(* Logix 5000 project; controller Line_Information_Standard vendor 1 type 14 code 151 rev 28.11; software revision 28.00 *)

TASK MainTask (continuous, watchdog 500 ms) : MainProgram

MODULES
   Local : vendor 1 type 14 code 151 (Compact 0, rev 28.11)
      Counters : Embedded (Compact 3, rev 1.1, Output RPI 20 ms)
      Analog_IO : Embedded (Compact 2, rev 1.1, Output RPI 80 ms)
      Discrete_IO : Embedded (Compact 1, rev 3.1, Output RPI 20 ms)
END_MODULES

TYPE ControlInterlock :   // Datatype for control interlocks to machines
STRUCT
   Connection : CONNECTION_STATUS;   // Machine connection status
   run : BOOL;   // OK to run machine
   jog : BOOL;   // OK to jog machine
   feed : BOOL;   // OK to feed machine
   commandRunSpeed : DINT;   // Commanded run speed
   commandJogSpeed : DINT;   // Commanded jog speed
   Time : DINT[7];   // Clock time
   MiscDINT : DINT[4];   // Miscellaneous digital values
   MiscREAL : REAL[4];   // Miscellaneous analog values
   MiscBOOL : BOOL[32];   // Miscellaneous bit values
END_STRUCT
END_TYPE

TYPE ConveyingControlInterlock :   // Datatype for control interlocks to conveying
STRUCT
   Connection : CONNECTION_STATUS;   // Machine connection status
   Running : BOOL[32];   // Machine running array
   Feeding : BOOL[32];   // Machine feeding array
   ProductIn : BOOL[32];   // Product in machine array
   CommandRunSpeed : DINT[64];   // Conveyor commanded run speed array
   Time : DINT[7];   // Clock time
   MiscDINT : DINT[8];   // Miscellaneous digital values
   MiscREAL : REAL[8];   // Miscellaneous analog values
   MiscBOOL : BOOL[64];   // Miscellaneous bit values
END_STRUCT
END_TYPE

TYPE ConveyingStatusInterlock :   // Datatype for status interlocks from conveying
STRUCT
   Connection : CONNECTION_STATUS;   // Machine connection status
   Faulted : BOOL[64];   // Conveyor faulted array
   Ready : BOOL[64];   // Conveyor ready array
   Running : BOOL[64];   // Conveyor running array
   Auto : BOOL[64];   // Conveyor in auto array
   Run : BOOL[32];   // OK to run machine array
   Feed : BOOL[32];   // OK to feed machine array
   ActualSpeed : DINT[64];   // Actual speed of conveyor array
   MiscDINT : DINT[8];   // Miscellaneous digital values
   MiscREAL : REAL[8];   // Miscellaneous analog values
   MiscBOOL : BOOL[64];   // Miscellaneous bit values
END_STRUCT
END_TYPE

TYPE LineInformation :   // Datatype for interfaces and displays
STRUCT
   Faults : BOOL[2048];   // Fault bit array
   MachineStatus : SINT[32];   // Machine statuses array
   MachineDown : BOOL[32];   // Machine down bit array
   BaseProductionCount : DINT[32];   // Base production counts array
   PackProductionCount : DINT[32];   // Package production counts array
   ActualBasePerPack : INT[32];   // Actual base per package multiplier array
   NominalBasePerPack : INT[32];   // Nominal base per package multiplier array
   ConveyorStatus : SINT[64];   // Conveyor statuses array
   Recipe : DINT[128];   // Recipe values
   Time : DINT[7];   // Clock time
   DST : SINT;   // Daylight saving time
   timeZone : SINT;   // Time zone UTC offset
   MiscDINT : DINT[8];   // Miscellaneous digital values
   MiscREAL : REAL[8];   // Miscellaneous analog values
   MiscBOOL : BOOL[64];   // Miscellaneous bit values
END_STRUCT
END_TYPE

TYPE MessageControlInterlock :   // Datatype for message control interlocks to machines
STRUCT
   Connection : SINT;   // Initial byte of memory to satisfy copy instruction
   run : BOOL;   // OK to run machine
   jog : BOOL;   // OK to jog machine
   feed : BOOL;   // OK to feed machine
   commandRunSpeed : DINT;   // Commanded run speed
   commandJogSpeed : DINT;   // Commanded jog speed
   Time : DINT[7];   // Clock time
   MiscDINT : DINT[4];   // Miscellaneous digital values
   MiscREAL : REAL[4];   // Miscellaneous analog values
   MiscBOOL : BOOL[32];   // Miscellaneous bit values
END_STRUCT
END_TYPE

TYPE MessageStatusInterlock :   // Datatype for message status interlocks from machines
STRUCT
   Connection : SINT;   // Initial byte of memory to satisfy copy instruction
   faulted : BOOL;   // Machine faulted
   ready : BOOL;   // Machine ready
   running : BOOL;   // Machine running
   jogging : BOOL;   // Machine jogging
   feeding : BOOL;   // Machine feeding
   productIn : BOOL;   // Product in machine
   actualSpeed : DINT;   // Actual speed of machine
   baseProductionCount : DINT;   // Base production count
   packProductionCount : DINT;   // Package production count
   basePerPack : INT;   // Base per package multiplier
   MiscDINT : DINT[4];   // Miscellaneous digital values
   MiscREAL : REAL[4];   // Miscellaneous analog values
   MiscBOOL : BOOL[32];   // Miscellaneous bit values
END_STRUCT
END_TYPE

TYPE StatusInterlock :   // Datatype for status interlocks from machines
STRUCT
   Connection : CONNECTION_STATUS;   // Machine connection status
   faulted : BOOL;   // Machine faulted
   ready : BOOL;   // Machine ready
   running : BOOL;   // Machine running
   jogging : BOOL;   // Machine jogging
   feeding : BOOL;   // Machine feeding
   productIn : BOOL;   // Product in machine
   actualSpeed : DINT;   // Actual speed of machine
   baseProductionCount : DINT;   // Base production count
   packProductionCount : DINT;   // Package production count
   basePerPack : INT;   // Base per package multiplier
   MiscDINT : DINT[4];   // Miscellaneous digital values
   MiscREAL : REAL[4];   // Miscellaneous analog values
   MiscBOOL : BOOL[32];   // Miscellaneous bit values
END_STRUCT
END_TYPE

VAR_GLOBAL   (* controller tags *)
   Clock : DINT[7] := ([0] := 2017, [1] := 4, [2] := 28, [3] := 22, [4] := 37, [5] := 15, [6] := 583819);   // Date and Time
        [0]   // Year
        [1]   // Month
        [2]   // Day
        [3]   // Hour
        [4]   // Minute
        [5]   // Second
        [6]   // Microsecond
   LineInformation : LineInformation := (Faults[17] := 1, Faults[353] := 1, Faults[2047] := 1, MachineStatus[0] := 3, MachineStatus[2] := 1, MachineStatus[3] := 2, MachineStatus[4] := 3, MachineStatus[5] := 4, MachineStatus[6] := 5, MachineStatus[9] := 6, BaseProductionCount[0] := 26905, BaseProductionCount[1] := 4706715, BaseProductionCount[2] := 13657446, BaseProductionCount[3] := 11278396, BaseProductionCount[4] := 7218001, BaseProductionCount[5] := 8116703, BaseProductionCount[6] := 30118, BaseProductionCount[7] := 29912, BaseProductionCount[8] := -2147453745, BaseProductionCount[9] := 30115, BaseProductionCount[10] := 29900, BaseProductionCount[11] := 29900, BaseProductionCount[12] := 29900, BaseProductionCount[13] := 29900, BaseProductionCount[14] := 29900, BaseProductionCount[15] := 29900, BaseProductionCount[16] := 29900, BaseProductionCount[17] := 29900, BaseProductionCount[18] := 29900, BaseProductionCount[19] := 29900, BaseProductionCount[20] := 29900, BaseProductionCount[21] := 29900, BaseProductionCount[22] := 29900, BaseProductionCount[23] := 29900, BaseProductionCount[24] := 29900, BaseProductionCount[25] := 29900, BaseProductionCount[26] := 29900, BaseProductionCount[27] := 29900, BaseProductionCount[28] := 29900, BaseProductionCount[29] := 29900, BaseProductionCount[30] := 29900, BaseProductionCount[31] := 29905, PackProductionCount[0] := 2990, PackProductionCount[1] := 2990, PackProductionCount[2] := 2990, PackProductionCount[3] := 2990, PackProductionCount[4] := 2990, PackProductionCount[5] := 2990, PackProductionCount[6] := 2990, PackProductionCount[7] := 2990, PackProductionCount[8] := 2990, PackProductionCount[9] := 2990, PackProductionCount[10] := 2990, PackProductionCount[11] := 2990, PackProductionCount[12] := 2990, PackProductionCount[13] := 2990, PackProductionCount[14] := 2990, PackProductionCount[15] := 2990, PackProductionCount[16] := 2990, PackProductionCount[17] := 2990,
        PackProductionCount[18] := 2990, PackProductionCount[19] := 2990, PackProductionCount[20] := 2990, PackProductionCount[21] := 2990, PackProductionCount[22] := 2990, PackProductionCount[23] := 2990, PackProductionCount[24] := 2990, PackProductionCount[25] := 2990, PackProductionCount[26] := 2990, PackProductionCount[27] := 2990, PackProductionCount[28] := 2990, PackProductionCount[29] := 2990, PackProductionCount[30] := 2990, PackProductionCount[31] := 2990, ActualBasePerPack[1] := 6, ActualBasePerPack[7] := 100, ActualBasePerPack[8] := 100, ActualBasePerPack[9] := 10, ActualBasePerPack[31] := 10, NominalBasePerPack[7] := 100, NominalBasePerPack[8] := 100, Recipe[0] := 641227448, Recipe[2] := 600, Recipe[3] := 700, Recipe[9] := 56, Recipe[15] := 25, Time[0] := 2017, Time[1] := 4, Time[2] := 28, Time[3] := 22, Time[4] := 37, DST := 1, timeZone := -7);
   ONS : BOOL[32];
   ONS01 : BOOL;
   pastDST : SINT := 1;   // Past state daylight savings time was sycronized
   PastTime : DINT[7] := ([0] := 2017, [1] := 4, [2] := 28, [3] := 22, [4] := 37);   // Past time the clock was sycronized
   pastTimeZone : SINT := -7;   // Past UTC offset time zone was syncronized
   Test : BOOL[32] := ([1] := 1, [2] := 1, [3] := 1);
   timeZoneStrings : STRING[6] := ([0] := 'UTC-05:00', [1] := 'UTC-06:00', [2] := 'UTC-07:00', [3] := 'UTC-08:00', [4] := 'UTC-09:00', [5] := 'UTC-10:00');   // Time zone
END_VAR

PROGRAM MainProgram   (* main routine MainRoutine *)

ROUTINE MainRoutine   (* ladder *)
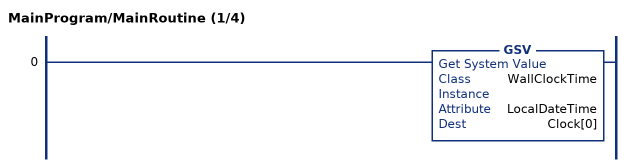
   0: GSV(WallClockTime,,LocalDateTime,Clock[0]);
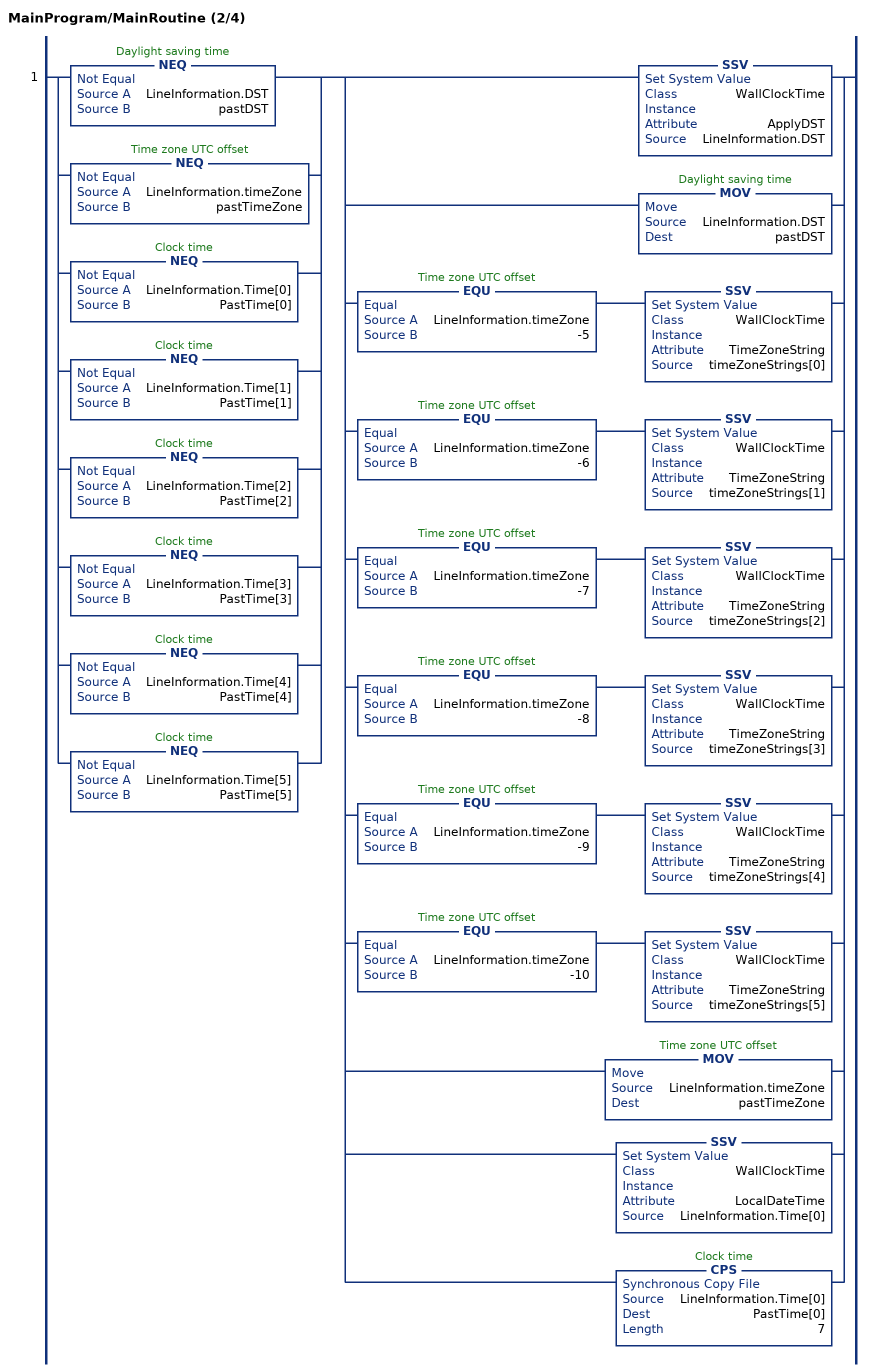
   1: [NEQ(LineInformation.DST,pastDST) ,NEQ(LineInformation.timeZone,pastTimeZone) ,NEQ(LineInformation.Time[0],PastTime[0]) ,NEQ(LineInformation.Time[1],PastTime[1]) ,NEQ(LineInformation.Time[2],PastTime[2]) ,NEQ(LineInformation.Time[3],PastTime[3]) ,NEQ(LineInformation.Time[4],PastTime[4]) ,NEQ(LineInformation.Time[5],PastTime[5]) ][SSV(WallClockTime,,ApplyDST,LineInformation.DST) ,MOV(LineInformation.DST,pastDST) ,EQU(LineInformation.timeZone,-5) SSV(WallClockTime,,TimeZoneString,timeZoneStrings[0]) ,EQU(LineInformation.timeZone,-6) SSV(WallClockTime,,TimeZoneString,timeZoneStrings[1]) ,EQU(LineInformation.timeZone,-7) SSV(WallClockTime,,TimeZoneString,timeZoneStrings[2]) ,EQU(LineInformation.timeZone,-8) SSV(WallClockTime,,TimeZoneString,timeZoneStrings[3]) ,EQU(LineInformation.timeZone,-9) SSV(WallClockTime,,TimeZoneString,timeZoneStrings[4]) ,EQU(LineInformation.timeZone,-10) SSV(WallClockTime,,TimeZoneString,timeZoneStrings[5]) ,MOV(LineInformation.timeZone,pastTimeZone) ,SSV(WallClockTime,,LocalDateTime,LineInformation.Time[0]) ,CPS(LineInformation.Time[0],PastTime[0],7) ];
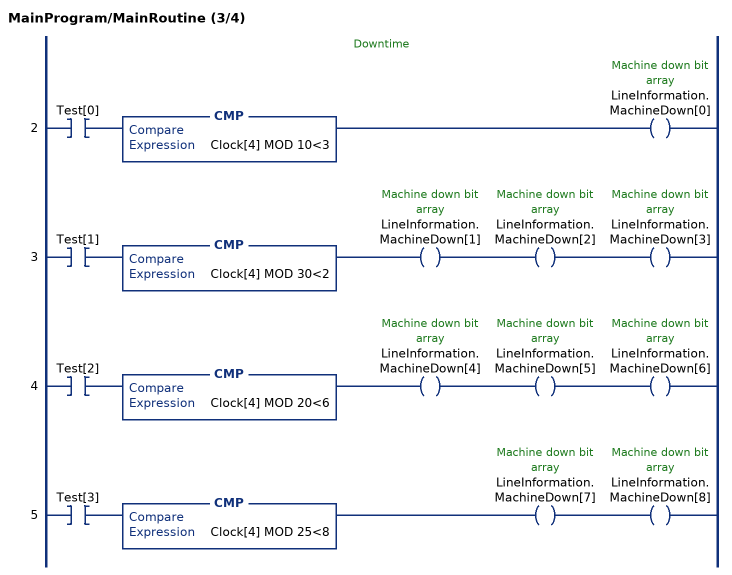
   // Downtime
   2: XIC(Test[0])CMP(Clock[4] MOD 10<3)OTE(LineInformation.MachineDown[0]);
   3: XIC(Test[1])CMP(Clock[4] MOD 30<2)OTE(LineInformation.MachineDown[1])OTE(LineInformation.MachineDown[2])OTE(LineInformation.MachineDown[3]);
   4: XIC(Test[2])CMP(Clock[4] MOD 20<6)OTE(LineInformation.MachineDown[4])OTE(LineInformation.MachineDown[5])OTE(LineInformation.MachineDown[6]);
   5: XIC(Test[3])CMP(Clock[4] MOD 25<8)OTE(LineInformation.MachineDown[7])OTE(LineInformation.MachineDown[8]);
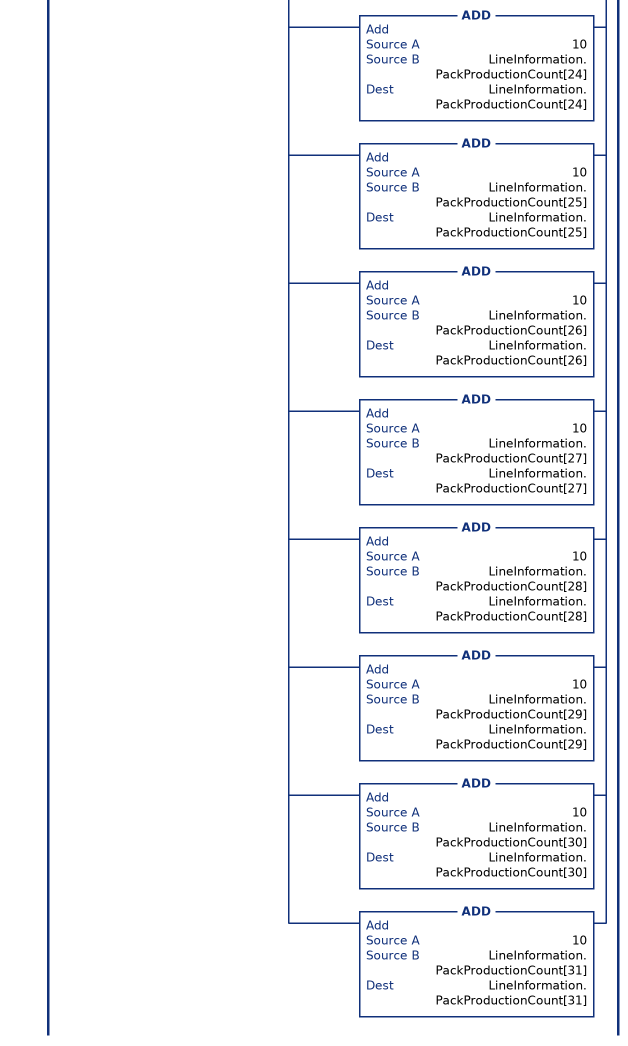
   6: XIC(Test[4])XIC(Clock[6].19)ONS(ONS01)[ADD(100,LineInformation.BaseProductionCount[0],LineInformation.BaseProductionCount[0]) ,ADD(100,LineInformation.BaseProductionCount[1],LineInformation.BaseProductionCount[1]) ,ADD(100,LineInformation.BaseProductionCount[2],LineInformation.BaseProductionCount[2]) ,ADD(100,LineInformation.BaseProductionCount[3],LineInformation.BaseProductionCount[3]) ,ADD(100,LineInformation.BaseProductionCount[4],LineInformation.BaseProductionCount[4]) ,ADD(100,LineInformation.BaseProductionCount[5],LineInformation.BaseProductionCount[5]) ,ADD(100,LineInformation.BaseProductionCount[6],LineInformation.BaseProductionCount[6]) ,ADD(100,LineInformation.BaseProductionCount[7],LineInformation.BaseProductionCount[7]) ,ADD(100,LineInformation.BaseProductionCount[8],LineInformation.BaseProductionCount[8]) ,ADD(100,LineInformation.BaseProductionCount[9],LineInformation.BaseProductionCount[9]) ,ADD(100,LineInformation.BaseProductionCount[10],LineInformation.BaseProductionCount[10]) ,ADD(100,LineInformation.BaseProductionCount[11],LineInformation.BaseProductionCount[11]) ,ADD(100,LineInformation.BaseProductionCount[12],LineInformation.BaseProductionCount[12]) ,ADD(100,LineInformation.BaseProductionCount[13],LineInformation.BaseProductionCount[13]) ,ADD(100,LineInformation.BaseProductionCount[14],LineInformation.BaseProductionCount[14]) ,ADD(100,LineInformation.BaseProductionCount[15],LineInformation.BaseProductionCount[15]) ,ADD(100,LineInformation.BaseProductionCount[16],LineInformation.BaseProductionCount[16]) ,ADD(100,LineInformation.BaseProductionCount[17],LineInformation.BaseProductionCount[17]) ,ADD(100,LineInformation.BaseProductionCount[18],LineInformation.BaseProductionCount[18]) ,ADD(100,LineInformation.BaseProductionCount[19],LineInformation.BaseProductionCount[19]) ,ADD(100,LineInformation.BaseProductionCount[20],LineInformation.BaseProductionCount[20]) ,ADD(100,LineInformation.BaseProductionCount[21],LineInformation.BaseProductionCount[21]) ,ADD(100,LineInformation.BaseProductionCount[22],LineInformation.BaseProductionCount[22]) ,ADD(100,LineInformation.BaseProductionCount[23],LineInformation.BaseProductionCount[23]) ,ADD(100,LineInformation.BaseProductionCount[24],LineInformation.BaseProductionCount[24]) ,ADD(100,LineInformation.BaseProductionCount[25],LineInformation.BaseProductionCount[25]) ,ADD(100,LineInformation.BaseProductionCount[26],LineInformation.BaseProductionCount[26]) ,ADD(100,LineInformation.BaseProductionCount[27],LineInformation.BaseProductionCount[27]) ,ADD(100,LineInformation.BaseProductionCount[28],LineInformation.BaseProductionCount[28]) ,ADD(100,LineInformation.BaseProductionCount[29],LineInformation.BaseProductionCount[29]) ,ADD(100,LineInformation.BaseProductionCount[30],LineInformation.BaseProductionCount[30]) ,ADD(100,LineInformation.BaseProductionCount[31],LineInformation.BaseProductionCount[31]) ,ADD(10,LineInformation.PackProductionCount[0],LineInformation.PackProductionCount[0]) ,ADD(10,LineInformation.PackProductionCount[1],LineInformation.PackProductionCount[1]) ,ADD(10,LineInformation.PackProductionCount[2],LineInformation.PackProductionCount[2]) ,ADD(10,LineInformation.PackProductionCount[3],LineInformation.PackProductionCount[3]) ,ADD(10,LineInformation.PackProductionCount[4],LineInformation.PackProductionCount[4]) ,ADD(10,LineInformation.PackProductionCount[5],LineInformation.PackProductionCount[5]) ,ADD(10,LineInformation.PackProductionCount[6],LineInformation.PackProductionCount[6]) ,ADD(10,LineInformation.PackProductionCount[7],LineInformation.PackProductionCount[7]) ,ADD(10,LineInformation.PackProductionCount[8],LineInformation.PackProductionCount[8]) ,ADD(10,LineInformation.PackProductionCount[9],LineInformation.PackProductionCount[9]) ,ADD(10,LineInformation.PackProductionCount[10],LineInformation.PackProductionCount[10]) ,ADD(10,LineInformation.PackProductionCount[11],LineInformation.PackProductionCount[11]) ,ADD(10,LineInformation.PackProductionCount[12],LineInformation.PackProductionCount[12]) ,ADD(10,LineInformation.PackProductionCount[13],LineInformation.PackProductionCount[13]) ,ADD(10,LineInformation.PackProductionCount[14],LineInformation.PackProductionCount[14]) ,ADD(10,LineInformation.PackProductionCount[15],LineInformation.PackProductionCount[15]) ,ADD(10,LineInformation.PackProductionCount[16],LineInformation.PackProductionCount[16]) ,ADD(10,LineInformation.PackProductionCount[17],LineInformation.PackProductionCount[17]) ,ADD(10,LineInformation.PackProductionCount[18],LineInformation.PackProductionCount[18]) ,ADD(10,LineInformation.PackProductionCount[19],LineInformation.PackProductionCount[19]) ,ADD(10,LineInformation.PackProductionCount[20],LineInformation.PackProductionCount[20]) ,ADD(10,LineInformation.PackProductionCount[21],LineInformation.PackProductionCount[21]) ,ADD(10,LineInformation.PackProductionCount[22],LineInformation.PackProductionCount[22]) ,ADD(10,LineInformation.PackProductionCount[23],LineInformation.PackProductionCount[23]) ,ADD(10,LineInformation.PackProductionCount[24],LineInformation.PackProductionCount[24]) ,ADD(10,LineInformation.PackProductionCount[25],LineInformation.PackProductionCount[25]) ,ADD(10,LineInformation.PackProductionCount[26],LineInformation.PackProductionCount[26]) ,ADD(10,LineInformation.PackProductionCount[27],LineInformation.PackProductionCount[27]) ,ADD(10,LineInformation.PackProductionCount[28],LineInformation.PackProductionCount[28]) ,ADD(10,LineInformation.PackProductionCount[29],LineInformation.PackProductionCount[29]) ,ADD(10,LineInformation.PackProductionCount[30],LineInformation.PackProductionCount[30]) ,ADD(10,LineInformation.PackProductionCount[31],LineInformation.PackProductionCount[31]) ];
END_ROUTINE
END_PROGRAM
